// SIMATIC S7-200 project (STEP 7-Micro/WIN), CPU 226 CN REL 02.01

ORGANIZATION_BLOCK 主程序:OB1
TITLE=项目信息：为庆丰630旋臂绞设备设计的绞线机控制系统，通过模拟量控制2个马达，实现多股细线均匀绞合。
// 设备信息：系统有编码器、变频器、主机和牵引马达。
// 程序注释：变频器模拟量输出将0-10VDC信号发送至变频器，精确控制主机马达和牵引马达的运行速度。
// 设备启动后，主机正转输出和主机反转输出根据操作需求驱动主机马达，并确保两者不可同时激活。主机运行时，线盘锁定输出在特定条件下置位，确保线盘固定，防止线材松动。此外，主机正转使能和主机反转使能依赖主机正转反馈和主机反转反馈的确认，确保马达状态与实际运行一致。
// 排线装置是绞线均匀性的关键。手动模式下，手动左移按钮或手动右移按钮触发排线左移输出或排线右移输出，实现排线控制。但排线左移输出和排线右移输出需满足左接近开关、右接近开关及相关禁止开关的条件，以保护设备运行范围。自动模式下，系统通过排位编码器A相输入和B相输入计算位置，并根据设定极限自动调整排线方向，确保线材排列整齐。
// 托板升降功能便于调整线盘高度以适应不同电缆生产。按下托板上升按钮时，托板上升输出置位，但需悬臂水平接近开关确认悬臂水平且托板下降按钮未按下。同样，托板下降按钮触发托板下降输出时，需确保悬臂水平、托板上升按钮未按下且托板下限制开关未检测到下极限，防止托板过度下降。
// 主机停止时，若主机转速低于1.0 RPM，悬臂刹车输出置位，稳住悬臂，防止滑动影响线材质量。紧急停止按钮、其他停止条件输入或托板下限制开关触发时，全机停止指示置位，确保工人和设备安全。
// 
BEGIN
Network 1 // 网络标题
// 网络注释
LD     SM0.1
CALL   Init:SBR6
?000
Network 2
LD     SM0.0
CALL   WinderSpeed:SBR2
CALL   ArrangeSpeed:SBR0
CALL   Logic:SBR3
CALL   Alarm:SBR4
CALL   Twi_Ins_Cal:SBR5
CALL   Output:SBR7
END_ORGANIZATION_BLOCK

SUBROUTINE_BLOCK ArrangeSpeed:SBR0
TITLE=子程序注释
BEGIN
Network 1 // 网络标题
// 收线编码器的减速链：
// N收=N编*36/100*80/48=0.3N编
// VD328:收线盘的速度
// N排正比于（N绞--N收）
// VD332：转速差
LD     SM0.0
MOVR   VD268, VD328
*R     0.3, VD328
MOVR   VD248, VD332
-R     VD328, VD332
Network 2
// 排线给定速度和N主，N收转速差的关系
// N排*螺距/排距=N主--N收
LD     SM0.0
LPS
ITD    VW118, VD340
AENO
DTR    VD340, VD344
LRD
MOVR   VD340, VD348
AENO
*R     VD332, VD348
AENO
MOVR   VD348, VD356
/R     VD352, VD356
LRD
MOVR   VD356, VD360
AENO
*R     32000.0, VD360
AENO
MOVR   VD360, VD364
/R     1460.0, VD364
LRD
MOVR   VD364, VD368
AENO
*R     10.0, VD368
AENO
MOVR   VD368, VD372
*R     1.2, VD372
LPP
ROUND  VD372, VD376
Network 3
// 排线位置信号清除
LD     SM0.0
LPS
A      I0.2
EU
=      M4.2
LPP
A      I0.5
EU
=      M4.3
Network 4
// 位置计算
// VD424:编码器圈数
// VD428:丝杆所转圈数
// VD432: 丝杆所走的MM数，即编码器第一次走到左接近开关时的位置。  标记为0MM处
// 5.0：丝杆导程
LDW>=  VW378, 100
LD     Q0.4
O      Q0.5
ALD
LPS
DTR    HC0, VD420
AENO
MOVR   VD420, VD424
/R     VD404, VD424
LPP
MOVR   VD424, VD428
AENO
/R     VD400, VD428
AENO
MOVR   VD428, VD436
*R     5.0, VD436
Network 5
// 左极限标记为0MM处
LD     M4.2
MOVR   0.0, VD432
MOVB   16#C0, SMB37
MOVD   0, SMD38
HSC    0
Network 6
// 0mm处的位置加上左位置设定为逻辑左限制(VD460) ，加上右位置为逻辑右限制(VD464) 
LD     SM0.0
LPS
ITD    VW122, VD440
AENO
DTR    VD440, VD444
LRD
ITD    VW124, VD450
AENO
DTR    VD450, VD454
LPP
MOVR   VD432, VD460
AENO
+R     VD444, VD460
AENO
MOVR   VD432, VD464
+R     VD454, VD464
Network 7
LD     SM0.0
LPS
AR<=   VD436, VD460
=      M4.4
LPP
AR>=   VD436, VD464
=      M4.5
END_SUBROUTINE_BLOCK

SUBROUTINE_BLOCK HMIdsp:SBR1
TITLE=子程序注释
BEGIN
Network 1 // 网络标题
// 网络注释
LD     SM0.0
LPS
ROUND  VD248, VD500
AENO
MOVW   VW502, VW100
LRD
ROUND  VD268, VD504
AENO
MOVW   VW506, VW102
LRD
ROUND  VD228, VD508
AENO
MOVW   VW510, VW104
LRD
MOVR   VD228, VD514
AENO
*R     1000.0, VD514
AENO
MOVR   VD514, VD518
/R     VD248, VD518
LPP
ROUND  VD518, VD522
AENO
MOVW   VW524, VW114
END_SUBROUTINE_BLOCK

SUBROUTINE_BLOCK WinderSpeed:SBR2
TITLE=子程序注释
BEGIN
Network 1 // 网络标题
// vw116:绞距设置
LD     SM0.0
LPS
ITD    VW116, VD300
AENO
DTR    VD300, VD304
LPP
MOVR   VD304, VD308
/R     1000.0, VD308
Network 2
// 线速度理论值，即PID给定值 
// vd312: 3-----120m/min,换算成0-10VDC给到变频的AI1
LD     SM0.0
LPS
MOVR   VD308, VD312
AENO
*R     VD248, VD312
AENO
MOVR   VD312, VD316
*R     32000.0, VD316
LRD
MOVR   VD316, VD320
AENO
/R     120.0, VD320
AENO
ROUND  VD320, VD324
LPP
MOVW   VW326, AQW0
Network 3
LD     M15.0
LPS
MOVR   VD308, VD600
AENO
*R     VD248, VD600
AENO
MOVR   VD600, VD604
/R     3.141459, VD604
LRD
MOVR   VD604, VD608
AENO
/R     0.3, VD608
AENO
MOVR   VD248, VD612
-R     VD608, VD612
LRD
MOVR   VD612, VD616
AENO
*R     32000.0, VD616
AENO
MOVR   VD616, VD620
/R     960.0, VD620
LPP
ROUND  VD620, VD624
AENO
MOVW   VW626, MW22
END_SUBROUTINE_BLOCK

SUBROUTINE_BLOCK Logic:SBR3
TITLE=子程序注释
BEGIN
Network 1 // 网络标题
// 主机S向,牵引S 向，自动时
LD     M0.7
AN     M2.6
LPS
A      M0.3
=      M3.1
LPP
AN     M0.3
=      M3.2
Network 2
// 包纸S 向， Z向
LD     M1.0
AN     M2.6
LPS
A      M0.4
=      M3.3
LPP
AN     M0.4
=      M3.4
Network 3
LD     I2.6
ED
R      M3.5, 1
Network 4
// 线盘锁定
LD     I2.6
EU
S      M3.5, 1
Network 5
// 托板上升控制
// I1.6:up
// i1.1:down
// i2.7: 悬臂水平接近
// I2.5：托板下限制
// Q1.6：up
// Q1.7：DOWN
LD     SM0.0
LPS
A      I1.6
A      I2.7
AN     I1.1
=      Q1.6
LPP
A      I1.1
A      I2.7
AN     I1.6
AN     I2.5
=      Q1.7
Network 6
// 排线控制
// 手动
// i0.7: <-------
// i1.0:------->
// M4.0:<--------
// M4.1:-------->
LDN    M2.6
LPS
A      I0.7
AN     I0.2
AN     I1.3
=      M4.0
LPP
A      I1.0
AN     I0.5
AN     I1.4
=      M4.1
Network 7
LD     M2.6
MOVB   0, MB5
Network 8
// 排线控制：自动,如果从来未启动过，MB5的位均OFF，先向左
// m5.0:<------------
LDN    M2.6
A      M0.7
EU
AB=    MB5, 0
O      M5.4
S      M5.0, 1
R      M5.4, 1
Network 9
// LEFT  DELAY
LD     M5.0
A      I0.2
S      M5.1, 1
R      M5.0, 1
Network 10
// ---------->M5.2
// 
LD     M5.1
TON    T101, 6
A      T101
S      M5.2, 1
R      M5.1, 1
Network 11
// RIGHT DELAY
LD     M5.2
A      I0.5
S      M5.3, 1
R      M5.2, 1
Network 12
// M5.4< ------
LD     M5.3
TON    T102, 6
A      T102
S      M5.4, 1
R      M5.3, 1
Network 13
// 悬臂刹车动作
LD     M0.7
ED
S      M6.0, 1
Network 14
LD     M6.0
AR>=   VD248, 0.0
AR<=   VD248, 1.0
=      M6.1
Network 15
LD     M0.7
EU
R      M6.0, 2
R      M3.5, 1
END_SUBROUTINE_BLOCK

SUBROUTINE_BLOCK Alarm:SBR4
TITLE=子程序注释
BEGIN
Network 1 // 网络标题
// 各种停机条件
LD     SM0.0
LPS
A      I1.5
=      M2.0
LRD
A      I2.0
=      M2.1
LRD
A      I1.3
=      M2.2
LPP
A      I1.4
=      M2.3
Network 2
// 全机停止
// I2.5: 托板限制
LD     M2.0
O      M2.1
O      M2.5
ON     I2.5
=      M2.6
Network 3
// 排线左向禁止
LD     M2.2
O      M2.6
O      I2.5
=      M2.7
Network 4
// 排线右向禁止
LD     M2.3
O      M2.6
=      M3.0
END_SUBROUTINE_BLOCK

SUBROUTINE_BLOCK Init:SBR6
TITLE=子程序注释
BEGIN
Network 1 // 网络标题
// 排位编码器，i0.0/i0.1.HSC0  MODE 9，SMB37，SMD38，SMD42。
LD     SM0.0
MOVB   16#FC, SMB37
MOVD   0, SMD38
MOVD   2147483647, SMD42
HDEF   0, 9
HSC    0
Network 2 // 网络标题
// 计米编码器，i0.3/i0.4.HSC4  MODE 9，SMB147，SMD148，SMD152。
LD     SM0.0
MOVB   16#FC, SMB157
MOVD   0, SMD158
MOVD   2147483647, SMD162
HDEF   5, 0
HSC    5
Network 3 // 网络标题
// 主机编码器i0.6 ，HSC1  MODE 0，SMB47，SMD48，SMD52。
LD     SM0.0
MOVB   16#F8, SMB47
MOVD   0, SMD48
MOVD   2147483647, SMD52
HDEF   1, 0
HSC    1
Network 4 // 网络标题
// 卷取i1.2 ，HSC2  MODE 0，SMB57，SMD58，SMD62。
LD     SM0.0
MOVB   16#F8, SMB57
MOVD   0, SMD58
MOVD   2147483647, SMD62
HDEF   2, 0
HSC    2
MOVB   200, SMB34
ATCH   INT_0:INT0, 10
ENI
END_SUBROUTINE_BLOCK

SUBROUTINE_BLOCK Output:SBR7
TITLE=子程序注释
BEGIN
Network 1 // 网络标题
// 网络注释
LD     SM0.0
LPS
A      M3.1
=      Q0.0
LRD
A      M3.2
=      Q0.1
LRD
LD     M3.1
LD     I2.1
AN     M3.1
AN     M3.2
OLD
ALD
=      Q0.2
LRD
LD     M3.2
LD     I2.2
AN     M3.1
AN     M3.2
OLD
ALD
=      Q0.3
LRD
LD     M5.2
O      M4.1
ALD
AN     I0.5
=      Q0.5
LRD
LD     M5.0
O      M5.4
O      M4.0
ALD
AN     I0.2
=      Q0.4
LRD
LPS
A      M3.3
=      Q0.7
LPP
A      M3.4
=      Q1.0
LRD
LD     M3.1
O      M3.2
ALD
=      Q1.1
LRD
LD     M3.3
O      M3.4
ALD
=      Q1.3
LRD
A      M2.6
=      Q1.5
LRD
LD     M6.1
O      M3.5
ALD
=      Q1.4
LPP
LD     M6.1
O      M3.5
ALD
=      Q1.2
END_SUBROUTINE_BLOCK

INTERRUPT_BLOCK INT_0:INT0
TITLE=中断程序注释
BEGIN
Network 1 // 网络标题
// 排位速度HC0 ，假定编码器为600PULSE/R
// 
// VD208: RPM
LDN    SM0.0
LPS
DTR    HC0, VD200
AENO
MOVR   VD200, VD204
/R     600.0, VD204
LRD
MOVR   VD204, VD208
*R     300.0, VD208
LRD
MOVB   16#C0, SMB37
LRD
MOVD   0, SMD38
LPP
HSC    0
Network 2 // 网络标题
// 线速HC4 ，假定编码器为600PULSE/R
// 
// VD228: RPM
LD     SM0.0
LPS
DTR    HC5, VD220
AENO
MOVR   VD220, VD224
/R     2000.0, VD224
LRD
MOVR   VD224, VD228
*R     300.0, VD228
LRD
MOVB   16#C0, SMB157
LRD
MOVD   0, SMD158
LPP
HSC    5
Network 3 // 网络标题
// 主机速度HC1，假定编码器为600PULSE/R
// 
// VD248: RPM
LD     SM0.0
LPS
DTR    HC1, VD240
AENO
MOVR   VD240, VD244
/R     600.0, VD244
LRD
MOVR   VD244, VD248
*R     300.0, VD248
LRD
MOVB   16#C0, SMB47
LRD
MOVD   0, SMD48
LPP
HSC    1
Network 4 // 网络标题
// 卷曲速度，假定编码器为600PULSE/R
// 
// VD268: RPM
LD     SM0.0
LPS
DTR    HC2, VD260
AENO
MOVR   VD260, VD264
/R     600.0, VD264
LRD
MOVR   VD264, VD268
*R     300.0, VD268
LRD
MOVB   16#C0, SMB57
LRD
MOVD   0, SMD58
LPP
HSC    2
END_INTERRUPT_BLOCK
